// TIA Portal V17 export
// export: Created 2022-07-28T18:02:46.4458702Z, ExportSetting None, DisplayName Totally Integrated Automation Portal, DisplayVersion V17, DisplayName TIA Portal Openness, DisplayVersion V17, DisplayName TIA Portal Teamcenter Gateway, DisplayVersion V17, DisplayName TIA Portal Version Control Interface, DisplayVersion V17, DisplayName TIA Portal Test Suite Advanced, DisplayVersion V17, DisplayName SINAMICS Startdrive Advanced, DisplayVersion V17, DisplayName SINAMICS DCC, DisplayVersion V17, DisplayName SINAMICS Startdrive G130, G150, S120, S150, SINAMICS MV, S210, DisplayVersion V17, DisplayName SINAMICS Startdrive G110M, G120, G120C, G120D, G120P, G115D, DisplayVersion V17, DisplayName STEP 7 Professional, DisplayVersion V17, DisplayName SIMATIC Energy Suite, DisplayVersion V17, DisplayName STEP 7 CFC, DisplayVersion V17, DisplayName STEP 7 Safety, DisplayVersion V17, DisplayName WinCC Advanced / Unified PC, DisplayVersion V17, DisplayName SIMATIC Visualization Architect, DisplayVersion V17
FUNCTION_BLOCK "Lib_FB_PID_Core"   // FB2, SCL
{ S7_Optimized_Access := 'TRUE' }
// stored: MemoryReserve 100, SetENOAutomatically false
   VAR_INPUT
      II_Obj_ID { ExternalAccessible := 'False'; ExternalVisible := 'False'; ExternalWritable := 'False'} : Int := -1;   // Tech ID of object
   END_VAR
   VAR_OUTPUT
      Q_DataErr { ExternalAccessible := 'False'; ExternalVisible := 'False'; ExternalWritable := 'False'} : Bool;   // 1 = Transfer data error occured (ObjDB -> temp, ect)
   END_VAR
   VAR
      s_PID { ExternalAccessible := 'False'; ExternalVisible := 'False'; ExternalWritable := 'False'} : PID_Compact;
      s_RampOut { S7_SetPoint := 'True'} : "Lib_FB_PT1_Ramp";
   END_VAR
   VAR_TEMP
      t_Obj_PIDCon : "Lib_UDT_PID_Core";
      tui_DB_ShiftPID : UInt;
      t_ObjAny_PIDCon : DB_ANY;
      t_ObjVar_PIDCon : Variant;
      ti_NumObjDB : UInt;   // Number of DB for storage object data
      t_DataErr : Bool;   // 1 = Transfer data error occured (ObjDB -> temp, ect)
      ti_Tmp : Int;
   END_VAR
   // s_PID.Mode := 4;
   // s_PID.RunModeByStartup := TRUE;
   // s_PID.SetSubstituteOutput := FALSE;
   // s_PID.ActivateRecoverMode := FALSE;
   // s_PID.Config.InputPerOn := FALSE;
   // s_PID.CycleTime.StartEstimation := false;
   // s_PID.CycleTime.EnEstimation := false;
   // s_PID.CycleTime.EnMonitoring := false;
   // s_PID.CtrlParamsBackUp.Cycle := 2.0;
   // s_PID.Retain.CtrlParams.Cycle := 0.1;
BEGIN
   REGION Read data
       #tui_DB_ShiftPID := "D_General_ProgramDATA".ui_Shift_DB_PID;
       #t_Obj_PIDCon := "D_ZeroTypes".PID_Core;

       //Read object data
       IF #II_Obj_ID >= 0
       THEN
           //Read PID data
           #ti_NumObjDB := INT_TO_UINT(#II_Obj_ID) + #tui_DB_ShiftPID;
           #t_ObjAny_PIDCon := UINT_TO_DB_ANY(#ti_NumObjDB);
           #t_ObjVar_PIDCon := DB_ANY_TO_VARIANT(in := #t_ObjAny_PIDCon, err => #ti_Tmp);

           //If DB exist and convertion without error
           IF #ti_Tmp = 0
           THEN
               VariantGet(SRC := #t_ObjVar_PIDCon,
                          DST => #t_Obj_PIDCon);
           ELSE
               #t_DataErr := true;
           END_IF;
       ELSE
           #t_DataErr := true;
       END_IF;
   END_REGION

   REGION Call PID

       #s_PID.Setpoint := #t_Obj_PIDCon.r_Setpoint;
       #s_PID.ManualValue := #t_Obj_PIDCon.r_ManualValue;
       #s_PID.Input := #t_Obj_PIDCon.r_Input;
       IF #t_Obj_PIDCon.ErrorAck
       THEN
           #s_PID.ErrorAck := #t_Obj_PIDCon.ErrorAck;
           #t_Obj_PIDCon.ErrorAck := false;
       END_IF;
       IF #t_Obj_PIDCon.Reset
       THEN
           #s_PID.Reset := true;
           #t_Obj_PIDCon.Reset := false;
       END_IF;
       #s_PID.Config.OutputUpperLimit := #t_Obj_PIDCon.r_OutputUpperLimit;
       #s_PID.Config.OutputLowerLimit := #t_Obj_PIDCon.r_OutputLowerLimit;
       #s_PID.CycleTime.Value := #t_Obj_PIDCon.r_CycleTime_Value;
       #s_PID.Retain.CtrlParams.Gain := #t_Obj_PIDCon.r_Gain;
       #s_PID.Retain.CtrlParams.Ti := #t_Obj_PIDCon.r_Ti;
       #s_PID.Retain.CtrlParams.Td := #t_Obj_PIDCon.r_Td;
       #s_PID.Config.InvertControl := #t_Obj_PIDCon.InvertControl;
       #s_PID.Config.SetpointUpperLimit := #t_Obj_PIDCon.r_SPUpperLimit;
       #s_PID.Config.SetpointLowerLimit := #t_Obj_PIDCon.r_SPLowerLimit;
       #s_PID.Config.InputUpperLimit := #t_Obj_PIDCon.r_PVUpperLimit;
       #s_PID.Config.InputLowerLimit := #t_Obj_PIDCon.r_PVLowerLimit;
       #s_PID.CtrlParamsBackUp.Cycle := #t_Obj_PIDCon.r_Cycle_PID;
       #s_PID.Mode := #t_Obj_PIDCon.i_Mode;
       IF #t_Obj_PIDCon.ModeActivate
       THEN
           #t_Obj_PIDCon.ModeActivate := false;
           #s_PID.ModeActivate := true;
       END_IF;

       IF #t_Obj_PIDCon.SetIntegralSum
       THEN
           //#t_Obj_PIDCon.SetIntegralSum := false;
           #s_PID.PIDCtrl.IntegralSum := #t_Obj_PIDCon.r_IntegralSum;
       END_IF;

       //Call PID
       #s_PID();

       IF #t_Obj_PIDCon.SetIntegralSum
       THEN
           #t_Obj_PIDCon.SetIntegralSum := false;
           #s_RampOut.ir_Input := #s_PID.Output;
           #s_RampOut.sr_Output := #s_PID.Output;
       END_IF;

       #s_RampOut(ir_Input := #s_PID.Output,
                  ir_T1_sec:=3.1,
                  ir_T_cycle_sec := #t_Obj_PIDCon.r_CycleTime_Value);

       #t_Obj_PIDCon.i_State := #s_PID.State;
       #t_Obj_PIDCon.Error := #s_PID.Error;
       #t_Obj_PIDCon.dw_ErrorBits := #s_PID.ErrorBits;
       #t_Obj_PIDCon.r_Output := #s_RampOut.qr_Output;
       IF NOT (#t_Obj_PIDCon.i_State = 3)
           AND NOT (#t_Obj_PIDCon.i_State = 4)
       THEN
           #t_Obj_PIDCon.r_Output := #t_Obj_PIDCon.r_OutputLowerLimit;
       END_IF;

       #t_Obj_PIDCon.OutPER := ABS(REAL_TO_INT(#s_RampOut.qr_Output/100.0*27648.0));
       #t_Obj_PIDCon.OutPWM := #s_PID.Output_PWM;

       #s_PID.ErrorAck := false;
       #s_PID.Reset := false;
       #s_PID.ModeActivate := false;

   END_REGION

   REGION Write data
       //DB num 
       IF #II_Obj_ID >= 0
           AND NOT #t_DataErr
       THEN
           //Write PID data
           VariantPut(SRC := #t_Obj_PIDCon,
                      DST := #t_ObjVar_PIDCon);
       ELSE
           #t_DataErr := true;
       END_IF;
   END_REGION

   #Q_DataErr := #t_DataErr;
END_FUNCTION_BLOCK
